// TIA Portal project "Soru3" (V15)

(* hardware
DEVICE "S7-1200 station_1"  S7-1200 Station
   slot 0: "Rack_0"  S7-1200 Rack  Rack  V1.0
   slot 1: "PLC_1"  CPU 1212C DC/DC/DC  6ES7 212-1AE40-0XB0  V4.2
*)

// ===== PLC "PLC_1"  CPU 1212C DC/DC/DC =====

VAR_GLOBAL   // PLC tag table "Default tag table"
   "Basla" AT %I0.1 : Bool;
   "Deger" AT %MD0 : DWord;
   "Motor_1" AT %Q0.0 : Bool;
   "Motor_2" AT %Q0.1 : Bool;
   "Dudur" AT %I0.0 : Bool;
END_VAR

// folder: System blocks/Program resources

DATA_BLOCK "Sayac"   // DB1
{ S7_Optimized_Access := 'TRUE' }
AUTHOR : Simatic
FAMILY : IEC
NAME : UCNTR
VERSION : 1.2
// stored: InstanceOfName IEC_UCOUNTER
"IEC_UCOUNTER"
BEGIN
END_DATA_BLOCK

// folder: (top level)

ORGANIZATION_BLOCK "Main"   // OB1, LAD, ProgramCycle
TITLE = "Main Program Sweep (Cycle)"
{ S7_Optimized_Access := 'TRUE' }
VERSION : 0.1
   VAR_INPUT
      Initial_Call : Bool;   // Initial call of this OB
      Remanence : Bool;   // =True, if remanent data are available
   END_VAR
BEGIN

REGION Network 1: Sayaç ayarlaması
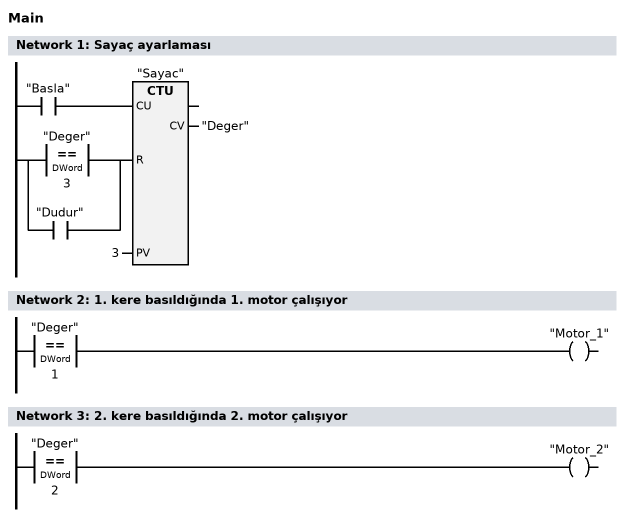
   "Sayac".CTU(CU := "Basla", R := ("Deger" = 3) OR "Dudur", PV := 3, CV => "Deger");
END_REGION

REGION Network 2: 1. kere basıldığında 1. motor çalışıyor
   RUNG wire#powerrail
      { S7_Templates := "SrcType := DWord" } EQ_Contact(in1 := "Deger", in2 := 1)
      Coil( "Motor_1" )
   END_RUNG
   // the same network as SCL:
   "Motor_1" := "Deger" = 1;
END_REGION

REGION Network 3: 2. kere basıldığında 2. motor çalışıyor
   RUNG wire#powerrail
      { S7_Templates := "SrcType := DWord" } EQ_Contact(in1 := "Deger", in2 := 2)
      Coil( "Motor_2" )
   END_RUNG
   // the same network as SCL:
   "Motor_2" := "Deger" = 2;
END_REGION
END_ORGANIZATION_BLOCK